FUNCTION_BLOCK FB_BalluffDevice
VAR_INPUT
END_VAR
VAR_OUTPUT
	Error	: BOOL;
	Position: REAL;
	Temperature	: REAL;
END_VAR
VAR
	Device	AT %I* : ST_BalluffDevice;
END_VAR

Error:= (Device.ErrorRegister<>0);
Temperature:= INT_TO_REAL(Device.Temperature);

END_FUNCTION_BLOCK

(* stored: Version 1.1.0.1, ProductVersion 3.1.4020.12
   POU FB_BalluffDevice: Id {50e9963e-f967-4f7e-8612-bce89c89f3ed}, SpecialFunc None *)
